FUNCTION ConvertPressure_Pirani : REAL
VAR_INPUT
	pressureInt : INT;
END_VAR
VAR
	voltage: REAL;
END_VAR

voltage :=  pressureInt / 3276.8;

IF voltage < 0.5 THEN
	ConvertPressure_Pirani := 1000; //ERROR (SENSOR DISCONNECTED??)
ELSE
	ConvertPressure_Pirani := EXPT(10, ( voltage - 6.143 ) / 1.286 ); // Converts ADC integer to mbars (formula from thermovac manual)
END_IF

END_FUNCTION

(* stored: Version 1.1.0.1, ProductVersion 3.1.4022.16
   POU ConvertPressure_Pirani: Id {2621c2f5-03e6-4670-936e-08e506e53fd5}, SpecialFunc None *)
